{attribute 'GeneratedUsingTerminal: KL6904-0001'}
{attribute addProperty BoxType "KL6904-0001"}
{attribute addProperty Id "StatusAT %I*BYTE0Register_InAT %I*UINT0Standard_QX_1AT %I*BYTE0Standard_QX_2AT %I*BYTE0Standard_QX_3AT %I*BYTE0Safety_QB_1AT %I*ARRAY[0..5] OF BYTE0Safety_QB_2AT %I*ARRAY[0..5] OF BYTE0Safety_QB_3AT %I*ARRAY[0..5] OF BYTE0Safety_QB_4AT %I*ARRAY[0..5] OF BYTE0Safety_QB_5AT %I*ARRAY[0..5] OF BYTE0Safety_QB_6AT %I*ARRAY[0..5] OF BYTE0Safety_QB_7AT %I*ARRAY[0..5] OF BYTE0Safety_QB_8AT %I*ARRAY[0..5] OF BYTE0Safety_QB_9AT %I*ARRAY[0..5] OF BYTE0Safety_QB_10AT %I*ARRAY[0..5] OF BYTE0Safety_QB_11AT %I*ARRAY[0..5] OF BYTE0Safety_QB_12AT %I*ARRAY[0..5] OF BYTE0Safety_QB_13AT %I*ARRAY[0..5] OF BYTE0Safety_QB_14AT %I*ARRAY[0..5] OF BYTE0Safety_QB_15AT %I*ARRAY[0..5] OF BYTE0ControlAT %Q*BYTE0Register_OutAT %Q*UINT0Standard_IX_1AT %Q*BYTE0Standard_IX_2AT %Q*BYTE0Standard_IX_3AT %Q*BYTE0Safety_IB_1AT %Q*ARRAY[0..5] OF BYTE0Safety_IB_2AT %Q*ARRAY[0..5] OF BYTE0Safety_IB_3AT %Q*ARRAY[0..5] OF BYTE0Safety_IB_4AT %Q*ARRAY[0..5] OF BYTE0Safety_IB_5AT %Q*ARRAY[0..5] OF BYTE0Safety_IB_6AT %Q*ARRAY[0..5] OF BYTE0Safety_IB_7AT %Q*ARRAY[0..5] OF BYTE0Safety_IB_8AT %Q*ARRAY[0..5] OF BYTE0Safety_IB_9AT %Q*ARRAY[0..5] OF BYTE0Safety_IB_10AT %Q*ARRAY[0..5] OF BYTE0Safety_IB_11AT %Q*ARRAY[0..5] OF BYTE0Safety_IB_12AT %Q*ARRAY[0..5] OF BYTE0Safety_IB_13AT %Q*ARRAY[0..5] OF BYTE0Safety_IB_14AT %Q*ARRAY[0..5] OF BYTE0Safety_IB_15AT %Q*ARRAY[0..5] OF BYTE0"}
{attribute addProperty CRC "4165648719"}
{attribute addProperty Size "0"}
TYPE Channel_F84AC14F :
STRUCT
	{attribute addProperty Name "Status"}
	Status AT %I* : BYTE;
	{attribute addProperty Name "Register_In"}
	Register_In AT %I* : UINT;
	{attribute addProperty Name "Standard_QX_1"}
	Standard_QX_1 AT %I* : BYTE;
	{attribute addProperty Name "Standard_QX_2"}
	Standard_QX_2 AT %I* : BYTE;
	{attribute addProperty Name "Standard_QX_3"}
	Standard_QX_3 AT %I* : BYTE;
	{attribute addProperty Name "Safety_QB_1"}
	Safety_QB_1 AT %I* : ARRAY[0..5] OF BYTE;
	{attribute addProperty Name "Safety_QB_2"}
	Safety_QB_2 AT %I* : ARRAY[0..5] OF BYTE;
	{attribute addProperty Name "Safety_QB_3"}
	Safety_QB_3 AT %I* : ARRAY[0..5] OF BYTE;
	{attribute addProperty Name "Safety_QB_4"}
	Safety_QB_4 AT %I* : ARRAY[0..5] OF BYTE;
	{attribute addProperty Name "Safety_QB_5"}
	Safety_QB_5 AT %I* : ARRAY[0..5] OF BYTE;
	{attribute addProperty Name "Safety_QB_6"}
	Safety_QB_6 AT %I* : ARRAY[0..5] OF BYTE;
	{attribute addProperty Name "Safety_QB_7"}
	Safety_QB_7 AT %I* : ARRAY[0..5] OF BYTE;
	{attribute addProperty Name "Safety_QB_8"}
	Safety_QB_8 AT %I* : ARRAY[0..5] OF BYTE;
	{attribute addProperty Name "Safety_QB_9"}
	Safety_QB_9 AT %I* : ARRAY[0..5] OF BYTE;
	{attribute addProperty Name "Safety_QB_10"}
	Safety_QB_10 AT %I* : ARRAY[0..5] OF BYTE;
	{attribute addProperty Name "Safety_QB_11"}
	Safety_QB_11 AT %I* : ARRAY[0..5] OF BYTE;
	{attribute addProperty Name "Safety_QB_12"}
	Safety_QB_12 AT %I* : ARRAY[0..5] OF BYTE;
	{attribute addProperty Name "Safety_QB_13"}
	Safety_QB_13 AT %I* : ARRAY[0..5] OF BYTE;
	{attribute addProperty Name "Safety_QB_14"}
	Safety_QB_14 AT %I* : ARRAY[0..5] OF BYTE;
	{attribute addProperty Name "Safety_QB_15"}
	Safety_QB_15 AT %I* : ARRAY[0..5] OF BYTE;
	{attribute addProperty Name "Control"}
	Control AT %Q* : BYTE;
	{attribute addProperty Name "Register_Out"}
	Register_Out AT %Q* : UINT;
	{attribute addProperty Name "Standard_IX_1"}
	Standard_IX_1 AT %Q* : BYTE;
	{attribute addProperty Name "Standard_IX_2"}
	Standard_IX_2 AT %Q* : BYTE;
	{attribute addProperty Name "Standard_IX_3"}
	Standard_IX_3 AT %Q* : BYTE;
	{attribute addProperty Name "Safety_IB_1"}
	Safety_IB_1 AT %Q* : ARRAY[0..5] OF BYTE;
	{attribute addProperty Name "Safety_IB_2"}
	Safety_IB_2 AT %Q* : ARRAY[0..5] OF BYTE;
	{attribute addProperty Name "Safety_IB_3"}
	Safety_IB_3 AT %Q* : ARRAY[0..5] OF BYTE;
	{attribute addProperty Name "Safety_IB_4"}
	Safety_IB_4 AT %Q* : ARRAY[0..5] OF BYTE;
	{attribute addProperty Name "Safety_IB_5"}
	Safety_IB_5 AT %Q* : ARRAY[0..5] OF BYTE;
	{attribute addProperty Name "Safety_IB_6"}
	Safety_IB_6 AT %Q* : ARRAY[0..5] OF BYTE;
	{attribute addProperty Name "Safety_IB_7"}
	Safety_IB_7 AT %Q* : ARRAY[0..5] OF BYTE;
	{attribute addProperty Name "Safety_IB_8"}
	Safety_IB_8 AT %Q* : ARRAY[0..5] OF BYTE;
	{attribute addProperty Name "Safety_IB_9"}
	Safety_IB_9 AT %Q* : ARRAY[0..5] OF BYTE;
	{attribute addProperty Name "Safety_IB_10"}
	Safety_IB_10 AT %Q* : ARRAY[0..5] OF BYTE;
	{attribute addProperty Name "Safety_IB_11"}
	Safety_IB_11 AT %Q* : ARRAY[0..5] OF BYTE;
	{attribute addProperty Name "Safety_IB_12"}
	Safety_IB_12 AT %Q* : ARRAY[0..5] OF BYTE;
	{attribute addProperty Name "Safety_IB_13"}
	Safety_IB_13 AT %Q* : ARRAY[0..5] OF BYTE;
	{attribute addProperty Name "Safety_IB_14"}
	Safety_IB_14 AT %Q* : ARRAY[0..5] OF BYTE;
	{attribute addProperty Name "Safety_IB_15"}
	Safety_IB_15 AT %Q* : ARRAY[0..5] OF BYTE;
END_STRUCT
END_TYPE

(* stored: Version 1.2.0.0, ProductVersion 3.1.4024.9
   DUT Channel_F84AC14F: Id {1779b162-75ee-4098-b1e4-e1c78f3cde33} *)
